FUNCTION_BLOCK UpdateSFC
VAR
	stSystemState	:	ST_Ledstrip_IOvars;
	r_SOC			:	REAL;
	r_Powerload		:	REAL;
	AnimationIndex: UINT;
END_VAR


VAR
	B_Update			: 	BOOL;
	ton_UpdateTimer		:	TON;
	ton_SOCUpdateTimer		:	TON;
	ton_AnimationUpdateTimer		:	TON;
	ftrig_Execute		:	f_trig;//TP := (PT := T#50MS);
	
	u_CurrentLEDColor		:	u_LedColor;
	
	FBRand	:	DRAND();
	seed	:	INT;
	
	Animation		:   UINT := 0;

	ChargeState		:	UINT;	//0=idle, 1=charging, 2=discharging
	
	st_Control		AT %Q*	:	stLedControl;
	st_Status		AT %I* :	stLedStatus;
	fTrig_CommandReady		:	f_trig;
	
	Param_AnimationLength			:	USINT		:=	5;
	Param_NrOfLeds					:	USINT 		:=	120;
	Param_UpdateInterval			:	TIME		:=	T#100MS;
	Param_AnimationUpdateInterval	:	TIME		:=	T#500MS;
	Param_SOCUpdateInterval			:	TIME		:=	T#1000MS;
	Param_EnablePowerLevel			:	BOOL		:=	TRUE;	
	params_CurrentTriggerlevel		:	INT			:=	10;
	by_LedIntensity					:	BYTE		:= 	127;
	
	UI_SOCLedIndex					: 	UINT;
	UI_PowerLevelIndex				:	UINT;
END_VAR

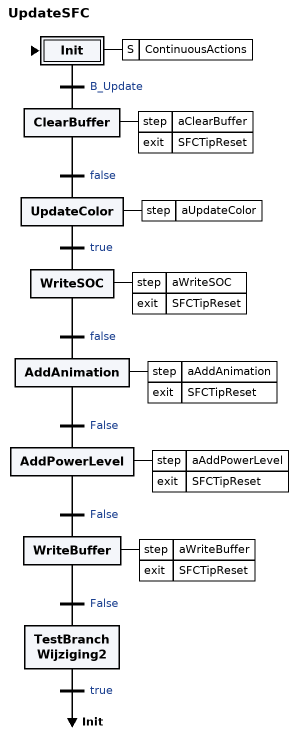
INITIAL_STEP Init:
    ContinuousActions(S);
END_STEP
TRANSITION FROM Init TO ClearBuffer
    := B_Update;
END_TRANSITION
STEP ClearBuffer:
    aClearBuffer(N);  // step action
    SFCTipReset(P0);  // exit action
END_STEP
TRANSITION FROM ClearBuffer TO UpdateColor
    := false;
END_TRANSITION
STEP UpdateColor:
    aUpdateColor(N);  // step action
END_STEP
TRANSITION FROM UpdateColor TO WriteSOC
    := true;
END_TRANSITION
STEP WriteSOC:
    aWriteSOC(N);  // step action
    SFCTipReset(P0);  // exit action
END_STEP
TRANSITION FROM WriteSOC TO AddAnimation
    := false;
END_TRANSITION
STEP AddAnimation:
    aAddAnimation(N);  // step action
    SFCTipReset(P0);  // exit action
END_STEP
TRANSITION FROM AddAnimation TO AddPowerLevel
    := False;
END_TRANSITION
STEP AddPowerLevel:
    aAddPowerLevel(N);  // step action
    SFCTipReset(P0);  // exit action
END_STEP
TRANSITION FROM AddPowerLevel TO WriteBuffer
    := False;
END_TRANSITION
STEP WriteBuffer:
    aWriteBuffer(N);  // step action
    SFCTipReset(P0);  // exit action
END_STEP
TRANSITION FROM WriteBuffer TO TestBranchWijziging2
    := False;
END_TRANSITION
STEP TestBranchWijziging2:
END_STEP
TRANSITION FROM TestBranchWijziging2 TO Init
    := true;
END_TRANSITION

ACTION aAddAnimation:

IF ChargeState = 0 THEN
	st_Control.b_Execute :=	FALSE;
	SFCTip := NOT SFCTip;
ELSE
	st_Control.by_Command := 1;
	st_Control.w_Index	:=	AnimationIndex;
	st_Control.w_Length	:=	1;
	st_Control.dw_Color :=  u_CurrentLEDColor.dw_LedColor;
	st_Control.b_Execute 	:=	NOT st_Control.b_Execute;
	
	IF ftrig_CommandReady.Q THEN
		st_Control.b_Execute :=	FALSE;
		SFCTip := TRUE;
	END_IF
END_IF
END_ACTION

ACTION aAddPowerLevel:
UI_PowerLevelIndex := LIMIT(1, REAL_TO_WORD((USINT_TO_REAL(Param_NrOfLeds)/100*r_Powerload)), USINT_TO_WORD(Param_NrOfLeds));

st_Control.by_Command := 1;
st_Control.w_Index	:=	UI_PowerLevelIndex;
st_Control.w_Length	:=	1;//UI_SOCLedIndex;
st_Control.dw_Color := 16#007F0000;
st_Control.b_Execute 	:=	NOT st_Control.b_Execute;

IF ftrig_CommandReady.Q THEN
	st_Control.b_Execute :=	FALSE;
	SFCTip := TRUE;
END_IF
END_ACTION

ACTION aClearBuffer:
b_update := FALSE;

st_Control.by_Command 	:= 	2;
st_Control.b_Execute 	:=	NOT st_Control.b_Execute;

IF ftrig_CommandReady.Q THEN
	st_Control.b_Execute :=	FALSE;
	SFCTip := TRUE;
END_IF

//testbrancheWijziging1
END_ACTION

ACTION aUpdateColor:

IF stSystemState.b_Error THEN
	u_CurrentLEDColor.st_LedColor.by_Red := by_LedIntensity;
	u_CurrentLEDColor.st_LedColor.by_Green := 0;
	u_CurrentLEDColor.st_LedColor.by_Blue := 0;
	u_CurrentLEDColor.st_LedColor.by_White := 0;
ELSIF stSystemState.b_warning THEN
	u_CurrentLEDColor.st_LedColor.by_Red := by_LedIntensity/2;
	u_CurrentLEDColor.st_LedColor.by_Green := by_LedIntensity/2;
	u_CurrentLEDColor.st_LedColor.by_Blue := 0;
	u_CurrentLEDColor.st_LedColor.by_White := 0;
ELSIF stSystemState.b_attention THEN
	u_CurrentLEDColor.st_LedColor.by_Red := 0;
	u_CurrentLEDColor.st_LedColor.by_Green := 0;
	u_CurrentLEDColor.st_LedColor.by_Blue := 0;
	u_CurrentLEDColor.st_LedColor.by_White := by_LedIntensity/2;	
ELSIF stSystemState.b_normal THEN
	u_CurrentLEDColor.st_LedColor.by_Red := 0;
	u_CurrentLEDColor.st_LedColor.by_Green := by_LedIntensity;
	u_CurrentLEDColor.st_LedColor.by_Blue := 0;
	u_CurrentLEDColor.st_LedColor.by_White := 0;
ELSE
	u_CurrentLEDColor.st_LedColor.by_Red := 0;
	u_CurrentLEDColor.st_LedColor.by_Green := 0;
	u_CurrentLEDColor.st_LedColor.by_Blue := by_LedIntensity;
	u_CurrentLEDColor.st_LedColor.by_White := 0;
END_IF
END_ACTION

ACTION aWriteBuffer:
st_Control.b_Update		:= TRUE;
st_Control.b_send		:= TRUE;
st_Control.b_Execute 	:=	NOT st_Control.b_Execute;

IF ftrig_CommandReady.Q THEN
	st_Control.b_Execute :=	FALSE;
	st_Control.b_Update		:= FALSE;
	st_Control.b_send		:= FALSE;
	SFCTip := TRUE;
END_IF
END_ACTION

ACTION aWriteSOC:
UI_SOCLedIndex := LIMIT(1, REAL_TO_WORD((USINT_TO_REAL(Param_NrOfLeds)/100*r_SOC)), USINT_TO_WORD(Param_NrOfLeds));

st_Control.by_Command := 1;
st_Control.w_Index	:=	0;
st_Control.w_Length	:=	UI_SOCLedIndex;
st_Control.dw_Color := u_CurrentLEDColor.dw_LedColor;
st_Control.b_Execute 	:=	NOT st_Control.b_Execute;

IF ftrig_CommandReady.Q THEN
	st_Control.b_Execute :=	FALSE;
	SFCTip := TRUE;
END_IF
END_ACTION

ACTION ContinuousActions:

ton_UpdateTimer(in := NOT ton_UpdateTimer.Q, PT := Param_UpdateInterval);

IF ton_UpdateTimer.Q THEN
	B_Update := TRUE;
END_IF

fTrig_CommandReady(Clk := st_Control.b_Execute);//st_Status.b_busy);

IF stSystemState.r_DCCurrent > params_CurrentTriggerlevel THEN
	ChargeState := 2;
ELSIF 	stSystemState.r_DCCurrent < (-params_CurrentTriggerlevel) THEN
	ChargeState := 1;
ELSE
	ChargeState := 0;
END_IF



ton_AnimationUpdateTimer(in := NOT ton_AnimationUpdateTimer.Q, PT := Param_AnimationUpdateInterval);
IF ton_AnimationUpdateTimer.q THEN
	CASE ChargeState OF
		0:
			AnimationIndex := UI_SOCLedIndex;// + Animation

			
		1: 
			IF AnimationIndex <= UI_SOCLedIndex THEN
				AnimationIndex := UI_SOCLedIndex + Param_AnimationLength-1;
				//Animation := Param_AnimationLength-1;
			ELSE
				AnimationIndex := AnimationIndex-1;
			END_IF
			
		2: 
			IF AnimationIndex >= UI_SOCLedIndex + Param_AnimationLength-1 THEN
				AnimationIndex := UI_SOCLedIndex;
			ELSE
				AnimationIndex := AnimationIndex+1;
			END_IF
	END_CASE
END_IF

FBRand(Seed := Seed);
ton_SOCUpdateTimer(in := NOT ton_SOCUpdateTimer.Q, PT := Param_SOCUpdateInterval);

IF ton_SOCUpdateTimer.Q THEN
	IF r_SOC < 0 THEN
		stSystemState.r_DCCurrent := -stSystemState.r_DCCurrent;
		r_SOC := 0;
	ELSIF r_SOC > 100 THEN
		stSystemState.r_DCCurrent := -stSystemState.r_DCCurrent;
		r_SOC := 100;
	ELSE
		r_SOC := r_SOC - (stSystemState.r_DCCurrent / (63 * 36));
	END_IF


	IF stSystemState.r_DCCurrent > 0 THEN
		stSystemState.r_DCCurrent := LIMIT(20, stSystemState.r_DCCurrent + ((FBRand.Num-0.5)*100), 630);
	ELSIF stSystemState.r_DCCurrent < 0 THEN
		stSystemState.r_DCCurrent := LIMIT(-630, stSystemState.r_DCCurrent + ((FBRand.Num-0.5)*100), -20);
	END_IF

	r_Powerload := ABS(stSystemState.r_DCCurrent/630)*100; 
	
END_IF
END_ACTION

ACTION SFCTipReset:
SFCTip := FALSE;
st_Control.b_Execute 	:= FALSE;
st_Control.b_Update		:= FALSE;
st_Control.b_send		:= FALSE;
END_ACTION

END_FUNCTION_BLOCK

(* stored: Version 1.1.0.1, ProductVersion 3.1.4024.12
   POU UpdateSFC: Id {f20a744b-1582-46ca-80fd-74156944d276}, SpecialFunc None
   Action aAddAnimation: Id {c6688011-423e-42a5-840d-8fe16380e42e}
   Action aAddPowerLevel: Id {549a9f18-3ecf-4676-b9e7-a0b20eeeab65}
   Action aClearBuffer: Id {0b7da1c8-afbc-4628-bd01-0bef2e3cc358}
   Action aUpdateColor: Id {4e76bdf7-6a20-4155-b939-5f89dc4a673d}
   Action aWriteBuffer: Id {cdc3b502-6001-4930-9808-6919dc75f559}
   Action aWriteSOC: Id {121aee4a-ce3a-4383-a6f2-d3460cb3782f}
   Action ContinuousActions: Id {81cf9bf6-bcba-47b3-b09a-4511abf179e8}
   Action SFCTipReset: Id {1426ff00-95c1-4f38-a242-fa54f3f7cf8a} *)
